Staubli VAL3: external.dtx

public aio aHeaterTime[2]
public aio aLight1[2]
public aio aLight2[2]
public aio aLight3[2]
public aio aState
public dio iCryoLongIn
public dio iCryoShortIn
public dio iEmergencyIn
public dio iFluor
public dio iFluorClosed
public dio iFluorOpen
public dio iGrip
public dio iGripClosed
public dio iGripOpen
public dio iHeaterStatus
public dio iIdent1
public dio iIdent2
public dio iIdent3
public dio iLevel1
public dio iLevel2
public dio iLevel3
public dio iLevel4
public dio iLevel5
public dio iLevelFault
public dio iLidClosed
public dio iPilatusPos
public dio iPlate1
public dio iPlate2
public dio iPlate3
public dio iPressureSensor
public dio iRack1
public dio iRack2
public dio iRack3
public dio iRack4
public dio iSampleStatus
public dio iSchock
public dio iTeste
public dio iTool
public dio oCryoLongOut
public dio oCryoShortOut
public dio oEmergencyOut
public dio oFluorDet
public dio oGripCmd
public dio oGripCmd2
public dio oHeater
public dio oLid
public dio oPilatusCover
public dio oResetFault
public dio oSample
public dio oShutter
public dio oVacuumValve
public mdesc mNomSpeed = {blend=off}
